// Mitsubishi GX Works2 project: 0715점프   PLC: Q02/Q02H

PROGRAM MAIN
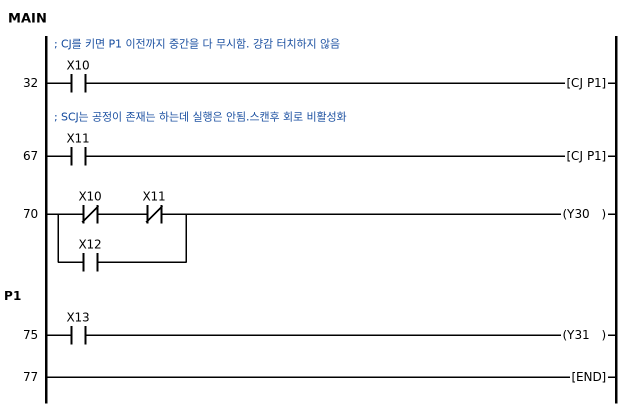
; CJ를 키면 P1 이전까지 중간을 다 무시함. 걍감 터치하지 않음
32    LD      X10
      CJ      P1
; SCJ는 공정이 존재는 하는데 실행은 안됨.스캔후 회로 비활성화
67    LD      X11
      SCJ     P1
70    LDI     X10
      ANI     X11
      OR      X12
      OUT     Y30
      P1
75    LD      X13
      OUT     Y31
77    END
END_PROGRAM
